{library PRIVATE}
(*
  Private Funtcion:
  Decode Status information messages.

*)
FUNCTION _GetStatusInformation : StatusInformationData
VAR_INPUT
	Data: 				DataGram;
END_VAR
VAR
END_VAR

_GetStatusInformation.Progress:=DWORD_TO_INT((SHR(Data.ParameterDW, 24) AND  16#FF));
_GetStatusInformation.FunctionNumber:=BYTE_TO_INT(Data.FunctionNumber);
_GetStatusInformation.ReturnValue:=BYTE_TO_INT(Data.FunctionType);
_GetStatusInformation.Extra:=BYTE_TO_INT(Data.ParameterB);

END_FUNCTION

(* stored: Version 1.1.0.1, ProductVersion 3.1.4024.2
   POU _GetStatusInformation: Id {2bf7c850-96f7-46b8-aaa9-54cf83b19e65}, SpecialFunc None *)
